(* Logix 5000 project; controller Safety vendor 1 type 14 code 86 rev 19.11; software revision 19.01; part 12 of 17 *)
(* tags used below, declared in another part *)
   A1_CoilCarSolPwrEn : BOOL;   // A1 UNW COIL CAR Solenoid Safe-Off Enable ( 1= Enable )
   A1_SolPwrEn : BOOL;   // A1 Solenoid Safe-Off Enable ( 1= Enable )
   A1_UnwLC_OK : BOOL;   // Unwind Light Curtain A/B ( 1= Not Blocked) ( 0= Blocked)
   A1_UnwLC_RstCmd : BOOL;   // Unwind Light Curtain Reset Command ( 1= Reset Cmd)
   C1_SolPwrEn : BOOL;   // C1 Solenoid Safe-Off Enable ( 1= Enable )
   CC_Toggle : DINT;   // TEST
   D1_SolPwrEn : BOOL;   // D1 Solenoid Safe-Off Enable ( 1= Enable )
   DPD_SolPwrEn : BOOL;   // DPD Solenoid Safe-Off Enable ( 1= Enable )
   E1_SolPwrEn : BOOL;   // E1 Solenoid Safe-Off Enable ( 1= Enable )
   Line_TotalMode : BOOL;   // Line TOTAL Mode ( 1= Total Mode) (0 = Coil to Coil)
   LineSts : UDT_SysStatus;
   OS4N_SolPwrEn : BOOL;   // OS4N Solenoid Safe-Off Enable ( 1= Enable )
   OS4S_SolPwrEn : BOOL;   // OS4S Solenoid Safe-Off Enable ( 1= Enable )
   PrCon_DrvsOff : BOOL;   // Product Conveyors (1-3) Drives OFF ( 1= OFF)
   PrCon_SafeTrqEn : BOOL;   // Product Conveyors Safe-Trq Off Enable ( 1= Enable )
   ScInCon_DrvsOff : BOOL;   // Scrap Incline Conveyor Drives OFF ( 1= OFF)
   ScInCon_SafeTrqEn : BOOL;   // Scrap Incline Conveyor Safe-Trq Off Enable ( 1= Enable )
   SDPLC_SolPwrEn : BOOL;   // SDPLC Solenoid Safe-Off Enable ( 1= Enable )
   ShearSts : UDT_ShearStatus;
   SkBkSt_DrvsOff : BOOL;   // Stacker Backstop Drives OFF ( 1= OFF)
   SkBkSt_SafeTrqEn : BOOL;   // Stacker Back Stop Safe-Trq Off Enable ( 1= Enable )
   SkBlwr_DrvsOff : BOOL;   // Stacker Blower Drives OFF ( 1= OFF)
   SkBlwr_SafeTrqEn : BOOL;   // Stacker Blower Safe-Trq Off Enable ( 1= Enable )
   Sr_DrvsOff : BOOL;   // Shear Pinch Roll/ Metering Back Up Drives OFF ( 1= OFF)
   Sr_SafeTrqEn : BOOL;   // Shear Pinch Roll/ Back Up Roll Safe-Trq Off Enable ( 1= Enable )
   SrCon_DrvsOff : BOOL;   // Shear Conveyor Drives OFF ( 1= OFF)
   SrCon_SafeTrqEn : BOOL;   // Shear Conveyor Safe-Trq Off Enable ( 1= Enable )
   StPR_DrvsOff : BOOL;   // Sheeter Pinch Roll Drives OFF ( 1= OFF)
   StPR_SafeTrqEn : BOOL;   // Sheeter Pinch Roll Safe-Trq Off Enable ( 1= Enable )
   UWCC_Rst_PB : ALIAS FOR SftyMap_Mach[0].10;   // Unwind Coil Car Safety Reset PB
   x406LCA047 : ALIAS FOR A1:21:I.Pt00Data;   // North/South Light Curtain Output A
   x406LCB052 : ALIAS FOR A1:21:I.Pt01Data;   // North/South Light Curtain Output B
   y172CR550 : ALIAS FOR SDPLC:2:O.Pt02Data;   // Line Soleniod Safe-Off
   y233CR040 : ALIAS FOR OS4N:5:O.Pt00Data;   // OS4N Solenoid Safe Off
   y243CR040 : ALIAS FOR OS4S:5:O.Pt00Data;   // OS4S Solenoid Safe Off
   y406CR050 : ALIAS FOR A1:20:O.Pt00Data;   // Line Solenoid Safe Off
   y406CR090 : ALIAS FOR A1:20:O.Pt01Data;   // Coil Car Solenoid Safe Off
   y435CR050 : ALIAS FOR C1:12:O.Pt00Data;   // Solenoid Safe Off
   y451CR050 : ALIAS FOR D1:12:O.Pt00Data;   // Soleniod Safe Off
   y464CR050 : ALIAS FOR E1:10:O.Pt00Data;   // Soleniod Safe Off
   y480CR050 : ALIAS FOR DPD:14:O.Pt00Data;   // Solenoid Safe Off
   y495CR050 : ALIAS FOR VS2:10:O.Pt00Data;   // Soleniod Safe Off
   y507CR090 : ALIAS FOR F1:19:O.Pt01Data;   // Rewind Coil Car Solenoid Safe Off
   y519CR050 : ALIAS FOR G1:11:O.Pt00Data;   // Line Solenoid Safe Off
   y533CR050 : ALIAS FOR H1:5:O.Pt00Data;   // Line Solenoid Safe Off
   y776MTR080SE : ALIAS FOR MCC4:3:O.Pt07Data;   // Shear Metering Backup Roll Safety Enable
   y776MTR080SP : ALIAS FOR MCC4:3:O.Pt06Data;   // Shear Metering Backup Roll Safety Power
   y779MTR080SE : ALIAS FOR MCC4:3:O.Pt01Data;   // Shear Pinch Roll Safety Enable
   y779MTR080SP : ALIAS FOR MCC4:3:O.Pt00Data;   // Shear Pinch Roll Safety Power
   y782MTR080SE : ALIAS FOR MCC4:3:O.Pt03Data;   // Sheeter Pinch Roll Safety Enable
   y782MTR080SP : ALIAS FOR MCC4:3:O.Pt02Data;   // Sheeter Pinch Roll Safety Power
   y785MTR080SE : ALIAS FOR MCC4:3:O.Pt05Data;   // Stacker Blower Safety Enable
   y785MTR080SP : ALIAS FOR MCC4:3:O.Pt04Data;   // Stacker Blower Safety Power
   y800MTR080SE : ALIAS FOR MCC5:3:O.Pt01Data;   // Scrap Incline Conveyor Safety Enable
   y800MTR080SP : ALIAS FOR MCC5:3:O.Pt00Data;   // Scrap Incline Conveyor Safety Power
   y804MTR080SE : ALIAS FOR MCC5:3:O.Pt03Data;   // Stacker Back Stop Safety Enable
   y804MTR080SP : ALIAS FOR MCC5:3:O.Pt02Data;   // Stacker Back Stop Safety Power
   y806MTR080SE : ALIAS FOR MCC5:3:O.Pt05Data;   // Product Conveyor 3 Safety Enable
   y806MTR080SP : ALIAS FOR MCC5:3:O.Pt04Data;   // Product Conveyor 3 Safety Power
   y808MTR080SE : ALIAS FOR MCC5:3:O.Pt07Data;   // Product Conveyor 1 Safety Enable
   y808MTR080SP : ALIAS FOR MCC5:3:O.Pt06Data;   // Product Conveyor 1 Safety Power
   y810MTR080SE : ALIAS FOR MCC5:4:O.Pt01Data;   // Product Conveyor 2 Safety Enable
   y810MTR080SP : ALIAS FOR MCC5:4:O.Pt00Data;   // Product Conveyor 2 Safety Power
   y812MTR080SE : ALIAS FOR MCC5:4:O.Pt03Data;   // Shear Conveyor Safety Enable
   y812MTR080SP : ALIAS FOR MCC5:4:O.Pt02Data;   // Shear Conveyor Safety Power
(* SafeOff, continued *)

ROUTINE B07_StPR_SafeTrqOff   (* ladder *)
// Sheeter Pinch Roll
// Safety Power Enable
// (Safe Trq Off and Drv Enable)
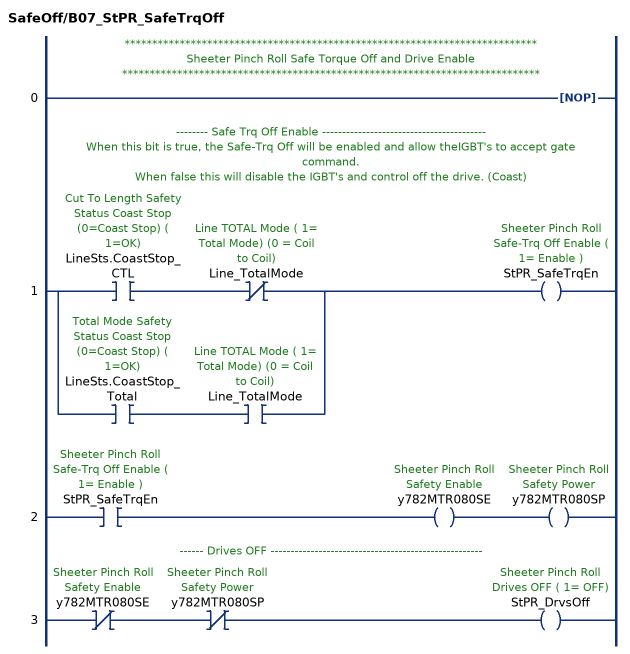
   // ***************************************************************************
   // Sheeter Pinch Roll Safe Torque Off and Drive Enable
   // ****************************************************************************
   0: NOP();
   // -------- Safe Trq Off Enable -----------------------------------------
   // When this bit is true, the Safe-Trq Off will be enabled and allow theIGBT's to accept gate command.
   // When false this will disable the IGBT's and control off the drive. (Coast)
   1: [XIC(LineSts.CoastStop_CTL) XIO(Line_TotalMode) ,XIC(LineSts.CoastStop_Total) XIC(Line_TotalMode) ]OTE(StPR_SafeTrqEn);
   2: XIC(StPR_SafeTrqEn)OTE(y782MTR080SE)OTE(y782MTR080SP);
   // ------ Drives OFF -----------------------------------------------------
   3: XIO(y782MTR080SE)XIO(y782MTR080SP)OTE(StPR_DrvsOff);
END_ROUTINE

ROUTINE B08_Sr_SafeTrqOff   (* ladder *)
// Sheear Pinch Roll /
// Back Up Metering
// Safety Power Enable
// (Safe Trq Off and Drv Enable)
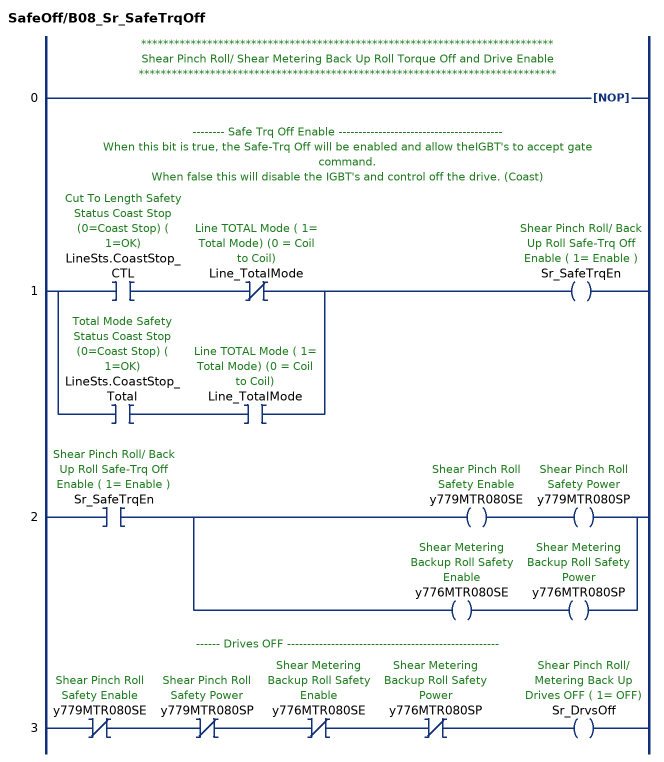
   // ***************************************************************************
   // Shear Pinch Roll/ Shear Metering Back Up Roll Torque Off and Drive Enable
   // ****************************************************************************
   0: NOP();
   // -------- Safe Trq Off Enable -----------------------------------------
   // When this bit is true, the Safe-Trq Off will be enabled and allow theIGBT's to accept gate command.
   // When false this will disable the IGBT's and control off the drive. (Coast)
   1: [XIC(LineSts.CoastStop_CTL) XIO(Line_TotalMode) ,XIC(LineSts.CoastStop_Total) XIC(Line_TotalMode) ]OTE(Sr_SafeTrqEn);
   2: XIC(Sr_SafeTrqEn)[OTE(y779MTR080SE) OTE(y779MTR080SP) ,OTE(y776MTR080SE) OTE(y776MTR080SP) ];
   // ------ Drives OFF -----------------------------------------------------
   3: XIO(y779MTR080SE)XIO(y779MTR080SP)XIO(y776MTR080SE)XIO(y776MTR080SP)OTE(Sr_DrvsOff);
END_ROUTINE

ROUTINE B09_SrCon_SafeTrqOff   (* ladder *)
// Shear Conveyor
// Safety Power Enable
// (Safe Trq Off and Drv Enable)
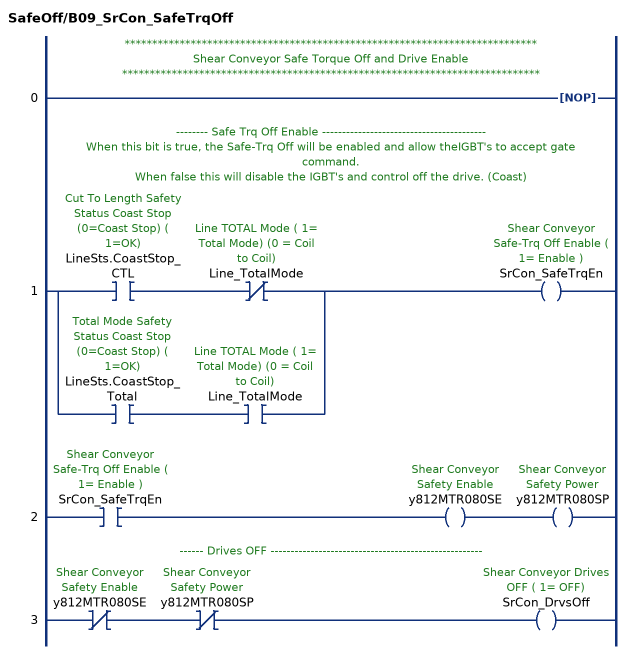
   // ***************************************************************************
   // Shear Conveyor Safe Torque Off and Drive Enable
   // ****************************************************************************
   0: NOP();
   // -------- Safe Trq Off Enable -----------------------------------------
   // When this bit is true, the Safe-Trq Off will be enabled and allow theIGBT's to accept gate command.
   // When false this will disable the IGBT's and control off the drive. (Coast)
   1: [XIC(LineSts.CoastStop_CTL) XIO(Line_TotalMode) ,XIC(LineSts.CoastStop_Total) XIC(Line_TotalMode) ]OTE(SrCon_SafeTrqEn);
   2: XIC(SrCon_SafeTrqEn)OTE(y812MTR080SE)OTE(y812MTR080SP);
   // ------ Drives OFF -----------------------------------------------------
   3: XIO(y812MTR080SE)XIO(y812MTR080SP)OTE(SrCon_DrvsOff);
END_ROUTINE

ROUTINE B10_PrCon_SafeTrqOff   (* ladder *)
// Product Conveyors (1-3)
// Safety Power Enable
// (Safe Trq Off and Drv Enable)
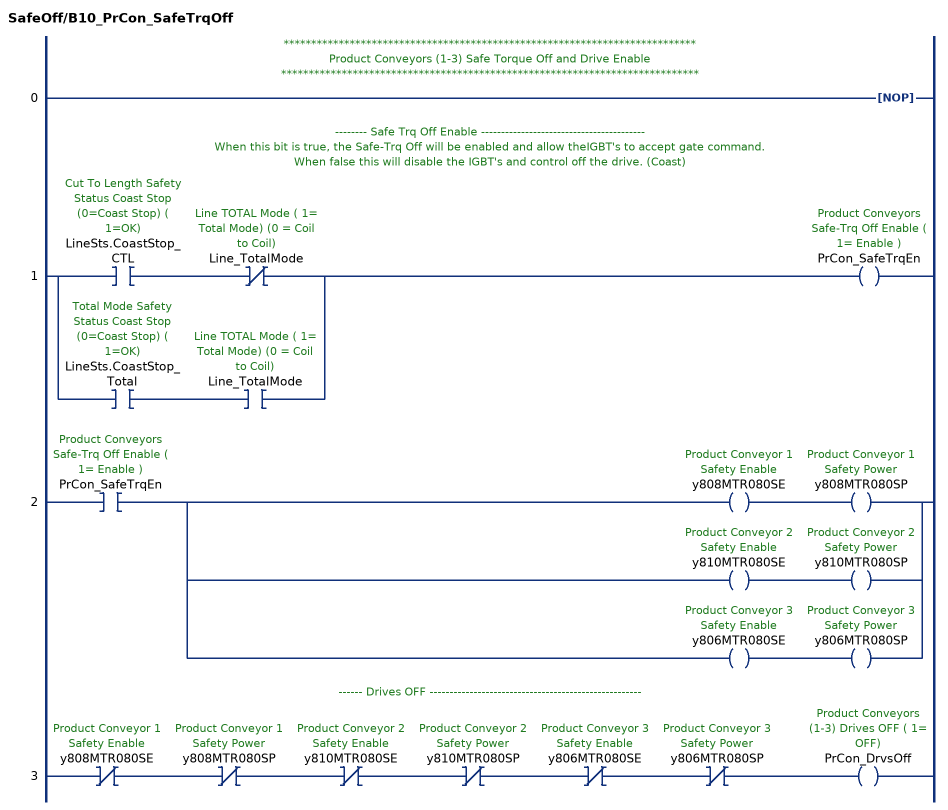
   // ***************************************************************************
   // Product Conveyors (1-3) Safe Torque Off and Drive Enable
   // ****************************************************************************
   0: NOP();
   // -------- Safe Trq Off Enable -----------------------------------------
   // When this bit is true, the Safe-Trq Off will be enabled and allow theIGBT's to accept gate command.
   // When false this will disable the IGBT's and control off the drive. (Coast)
   1: [XIC(LineSts.CoastStop_CTL) XIO(Line_TotalMode) ,XIC(LineSts.CoastStop_Total) XIC(Line_TotalMode) ]OTE(PrCon_SafeTrqEn);
   2: XIC(PrCon_SafeTrqEn)[OTE(y808MTR080SE) OTE(y808MTR080SP) ,OTE(y810MTR080SE) OTE(y810MTR080SP) ,OTE(y806MTR080SE) OTE(y806MTR080SP) ];
   // ------ Drives OFF -----------------------------------------------------
   3: XIO(y808MTR080SE)XIO(y808MTR080SP)XIO(y810MTR080SE)XIO(y810MTR080SP)XIO(y806MTR080SE)XIO(y806MTR080SP)OTE(PrCon_DrvsOff);
END_ROUTINE

ROUTINE B11_ScIncCon_SafeTrqOff   (* ladder *)
// Scrap Incline Conveyor
// Safety Power Enable
// (Safe Trq Off and Drv Enable)
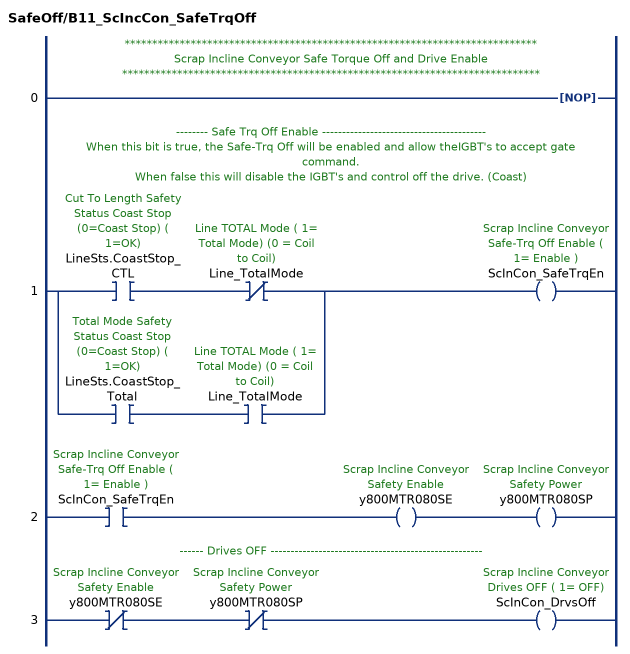
   // ***************************************************************************
   // Scrap Incline Conveyor Safe Torque Off and Drive Enable
   // ****************************************************************************
   0: NOP();
   // -------- Safe Trq Off Enable -----------------------------------------
   // When this bit is true, the Safe-Trq Off will be enabled and allow theIGBT's to accept gate command.
   // When false this will disable the IGBT's and control off the drive. (Coast)
   1: [XIC(LineSts.CoastStop_CTL) XIO(Line_TotalMode) ,XIC(LineSts.CoastStop_Total) XIC(Line_TotalMode) ]OTE(ScInCon_SafeTrqEn);
   2: XIC(ScInCon_SafeTrqEn)OTE(y800MTR080SE)OTE(y800MTR080SP);
   // ------ Drives OFF -----------------------------------------------------
   3: XIO(y800MTR080SE)XIO(y800MTR080SP)OTE(ScInCon_DrvsOff);
END_ROUTINE

ROUTINE B12_SkBlwr_SafeTrqOff   (* ladder *)
// Stacker Blower
// Safety Power Enable
// (Safe Trq Off and Drv Enable)
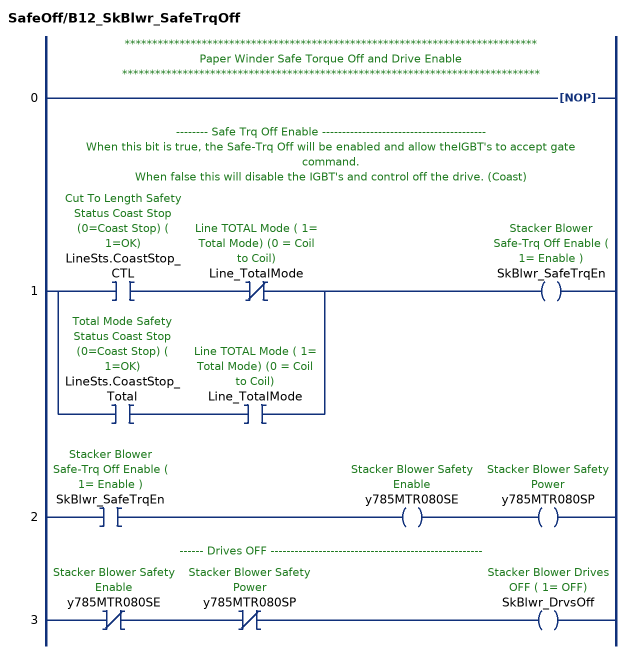
   // ***************************************************************************
   // Paper Winder Safe Torque Off and Drive Enable
   // ****************************************************************************
   0: NOP();
   // -------- Safe Trq Off Enable -----------------------------------------
   // When this bit is true, the Safe-Trq Off will be enabled and allow theIGBT's to accept gate command.
   // When false this will disable the IGBT's and control off the drive. (Coast)
   1: [XIC(LineSts.CoastStop_CTL) XIO(Line_TotalMode) ,XIC(LineSts.CoastStop_Total) XIC(Line_TotalMode) ]OTE(SkBlwr_SafeTrqEn);
   2: XIC(SkBlwr_SafeTrqEn)OTE(y785MTR080SE)OTE(y785MTR080SP);
   // ------ Drives OFF -----------------------------------------------------
   3: XIO(y785MTR080SE)XIO(y785MTR080SP)OTE(SkBlwr_DrvsOff);
END_ROUTINE

ROUTINE B13_SkBkSt_SafeTrqOff   (* ladder *)
// Stacker Back Stop
// Safety Power Enable
// (Safe Trq Off and Drv Enable)
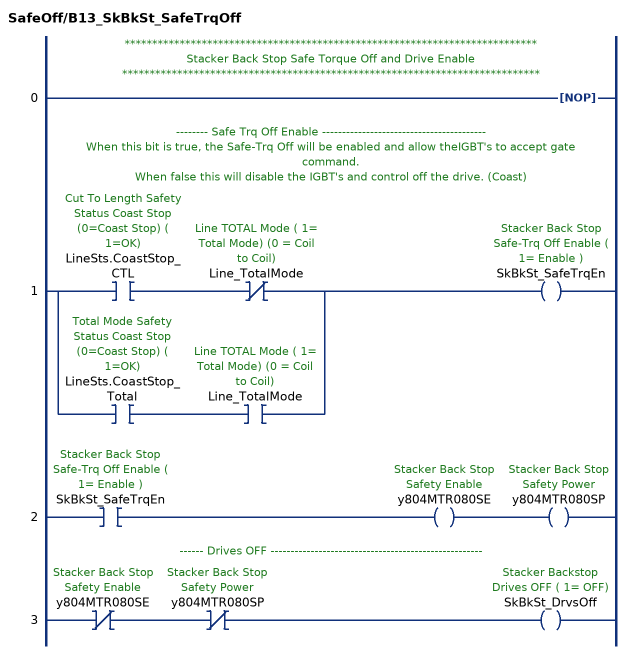
   // ***************************************************************************
   // Stacker Back Stop Safe Torque Off and Drive Enable
   // ****************************************************************************
   0: NOP();
   // -------- Safe Trq Off Enable -----------------------------------------
   // When this bit is true, the Safe-Trq Off will be enabled and allow theIGBT's to accept gate command.
   // When false this will disable the IGBT's and control off the drive. (Coast)
   1: [XIC(LineSts.CoastStop_CTL) XIO(Line_TotalMode) ,XIC(LineSts.CoastStop_Total) XIC(Line_TotalMode) ]OTE(SkBkSt_SafeTrqEn);
   2: XIC(SkBkSt_SafeTrqEn)OTE(y804MTR080SE)OTE(y804MTR080SP);
   // ------ Drives OFF -----------------------------------------------------
   3: XIO(y804MTR080SE)XIO(y804MTR080SP)OTE(SkBkSt_DrvsOff);
END_ROUTINE
END_PROGRAM

PROGRAM Safety_JUNK   (* main routine Scratch *)

ROUTINE Scratch   (* ladder *)
   0: NOP();
END_ROUTINE
END_PROGRAM

PROGRAM Solenoid_Pwr   (* main routine A00_Main *)
// Control fo the Field Power
// to the Solenoids

ROUTINE A00_Main   (* ladder *)
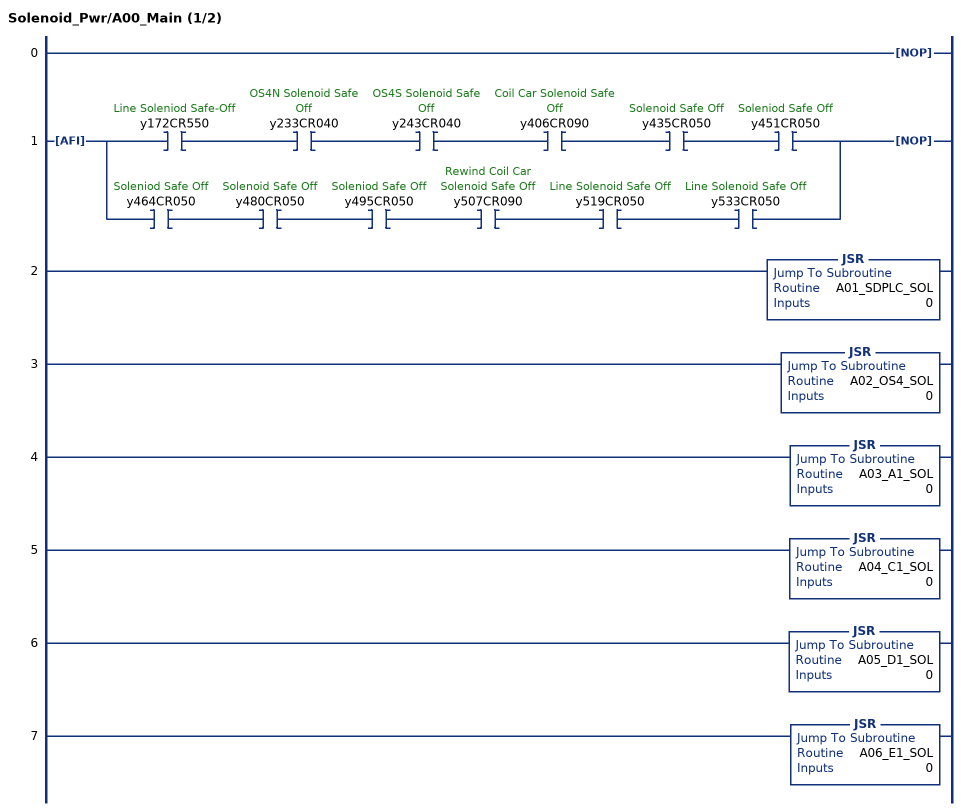
   0: NOP();
   1: AFI()[XIC(y172CR550) XIC(y233CR040) XIC(y243CR040) XIC(y406CR090) XIC(y435CR050) XIC(y451CR050) ,XIC(y464CR050) XIC(y480CR050) XIC(y495CR050) XIC(y507CR090) XIC(y519CR050) XIC(y533CR050) ]NOP();
   2: JSR(A01_SDPLC_SOL,0);
   3: JSR(A02_OS4_SOL,0);
   4: JSR(A03_A1_SOL,0);
   5: JSR(A04_C1_SOL,0);
   6: JSR(A05_D1_SOL,0);
   7: JSR(A06_E1_SOL,0);
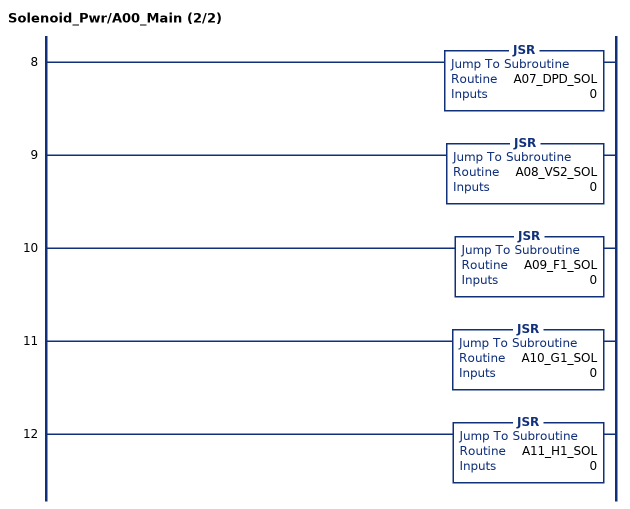
   8: JSR(A07_DPD_SOL,0);
   9: JSR(A08_VS2_SOL,0);
   10: JSR(A09_F1_SOL,0);
   11: JSR(A10_G1_SOL,0);
   12: JSR(A11_H1_SOL,0);
END_ROUTINE

ROUTINE A01_SDPLC_SOL   (* ladder *)
// SDPLC
// Solenoid Power Enable
// (FPD Power Removal)
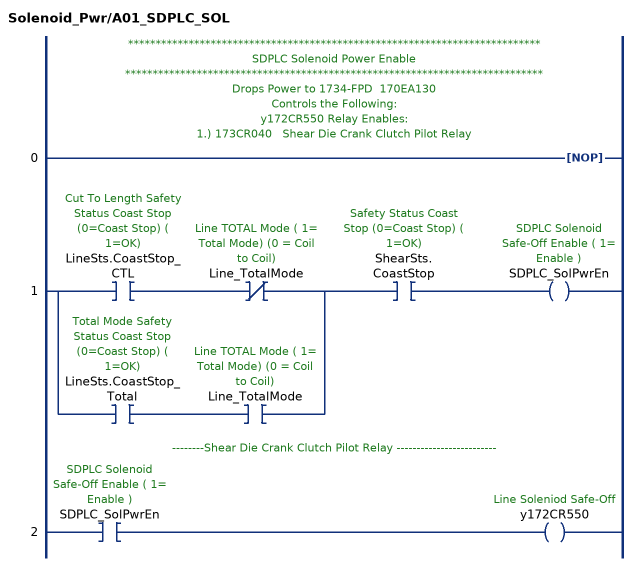
   // ***************************************************************************
   // SDPLC Solenoid Power Enable
   // ****************************************************************************
   // Drops Power to 1734-FPD	170EA130
   // Controls the Following:
   // y172CR550 Relay Enables:
   // 1.) 173CR040   Shear Die Crank Clutch Pilot Relay
   0: NOP();
   1: [XIC(LineSts.CoastStop_CTL) XIO(Line_TotalMode) ,XIC(LineSts.CoastStop_Total) XIC(Line_TotalMode) ]XIC(ShearSts.CoastStop)OTE(SDPLC_SolPwrEn);
   // --------Shear Die Crank Clutch Pilot Relay -------------------------
   2: XIC(SDPLC_SolPwrEn)OTE(y172CR550);
END_ROUTINE

ROUTINE A02_OS4_SOL   (* ladder *)
// OS4N/S
// Solenoid Power Enable
// (FPD Power Removal)
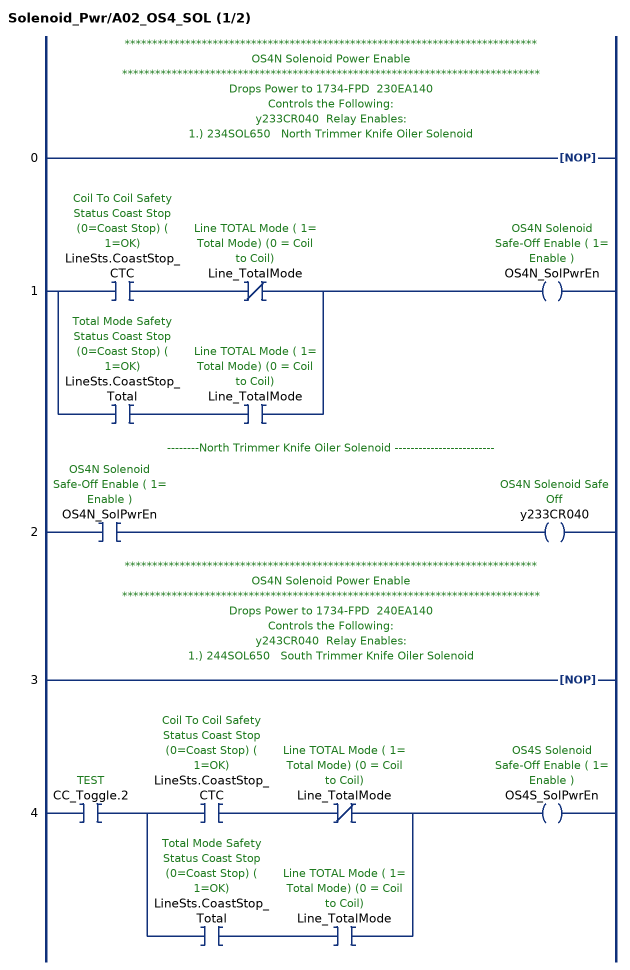
   // ***************************************************************************
   // OS4N Solenoid Power Enable
   // ****************************************************************************
   // Drops Power to 1734-FPD	230EA140
   // Controls the Following:
   // y233CR040  Relay Enables:
   // 1.) 234SOL650   North Trimmer Knife Oiler Solenoid
   0: NOP();
   1: [XIC(LineSts.CoastStop_CTC) XIO(Line_TotalMode) ,XIC(LineSts.CoastStop_Total) XIC(Line_TotalMode) ]OTE(OS4N_SolPwrEn);
   // --------North Trimmer Knife Oiler Solenoid -------------------------
   2: XIC(OS4N_SolPwrEn)OTE(y233CR040);
   // ***************************************************************************
   // OS4N Solenoid Power Enable
   // ****************************************************************************
   // Drops Power to 1734-FPD	240EA140
   // Controls the Following:
   // y243CR040  Relay Enables:
   // 1.) 244SOL650   South Trimmer Knife Oiler Solenoid
   3: NOP();
   4: XIC(CC_Toggle.2)[XIC(LineSts.CoastStop_CTC) XIO(Line_TotalMode) ,XIC(LineSts.CoastStop_Total) XIC(Line_TotalMode) ]OTE(OS4S_SolPwrEn);
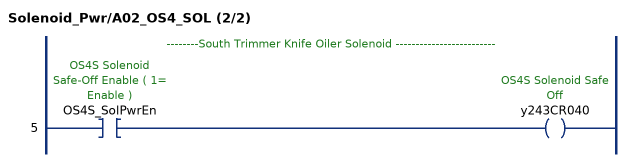
   // --------South Trimmer Knife Oiler Solenoid -------------------------
   5: XIC(OS4S_SolPwrEn)OTE(y243CR040);
END_ROUTINE

ROUTINE A03_A1_SOL   (* ladder *)
// A1
// Solenoid Power Enable
// (FPD Power Removal)
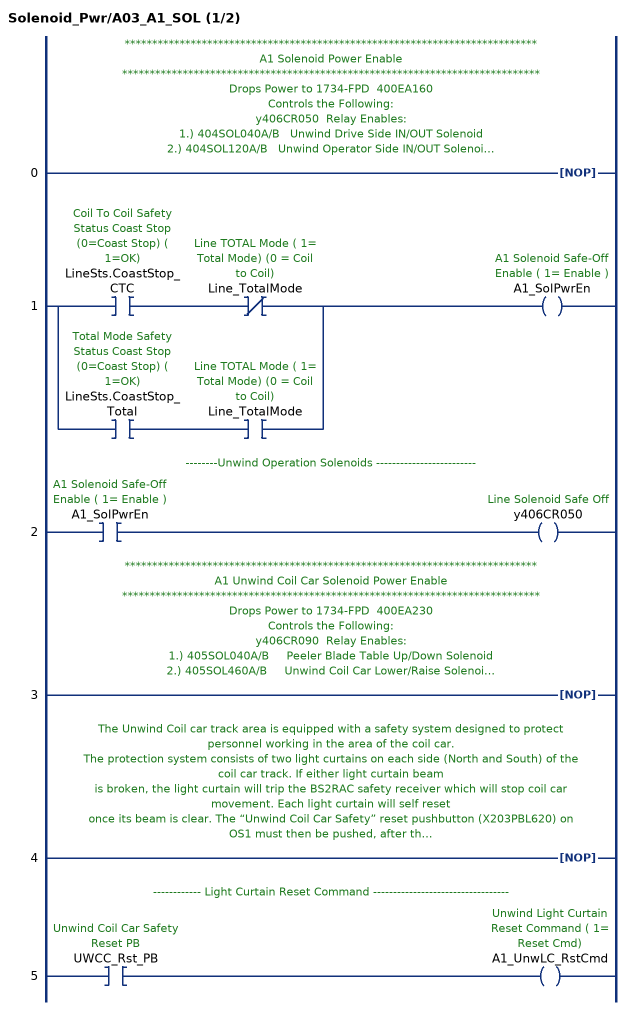
   // ***************************************************************************
   // A1 Solenoid Power Enable
   // ****************************************************************************
   // Drops Power to 1734-FPD	400EA160
   // Controls the Following:
   // y406CR050  Relay Enables:
   // 1.) 404SOL040A/B   Unwind Drive Side IN/OUT Solenoid
   // 2.) 404SOL120A/B   Unwind Operator Side IN/OUT Solenoid
   // 3.) 404SOL220A/B   Unwind Reel Tandem North Solenoid
   // 4.) 404SOL300         Unwind Reel Tandem Unlock Solenoid
   // 5.) 404SOL460A      Unwind Hold Down Roll Lower/Raise Solenoid
   // 6.) 404SOL640A/B   Unwind Peeler Blade Extend/Retract Solenoid
   // 7.) 404SOL680A/B   Unwind Peeler Blade Pivot Lower/Raise Solenoid
   0: NOP();
   1: [XIC(LineSts.CoastStop_CTC) XIO(Line_TotalMode) ,XIC(LineSts.CoastStop_Total) XIC(Line_TotalMode) ]OTE(A1_SolPwrEn);
   // --------Unwind Operation Solenoids -------------------------
   2: XIC(A1_SolPwrEn)OTE(y406CR050);
   // ***************************************************************************
   // A1 Unwind Coil Car Solenoid Power Enable
   // ****************************************************************************
   // Drops Power to 1734-FPD	400EA230
   // Controls the Following:
   // y406CR090  Relay Enables:
   // 1.) 405SOL040A/B     Peeler Blade Table Up/Down Solenoid
   // 2.) 405SOL460A/B     Unwind Coil Car Lower/Raise Solenoid
   // 3.) 405SOL540A/B     Unwind Coil Car Traverse IN/OUT Solenoid
   3: NOP();
   // The Unwind Coil car track area is equipped with a safety system designed to protect personnel working in the area of the coil car.
   // The protection system consists of two light curtains on each side (North and South) of the coil car track. If either light curtain beam
   // is broken, the light curtain will trip the BS2RAC safety receiver which will stop coil car movement. Each light curtain will self reset
   //  once its beam is clear. The “Unwind Coil Car Safety” reset pushbutton (X203PBL620) on OS1 must then be pushed, after the
   // area has been cleared, to reset the system and allow the coil car to continue movement.
   4: NOP();
   // ------------ Light Curtain Reset Command ----------------------------------
   5: XIC(UWCC_Rst_PB)OTE(A1_UnwLC_RstCmd);
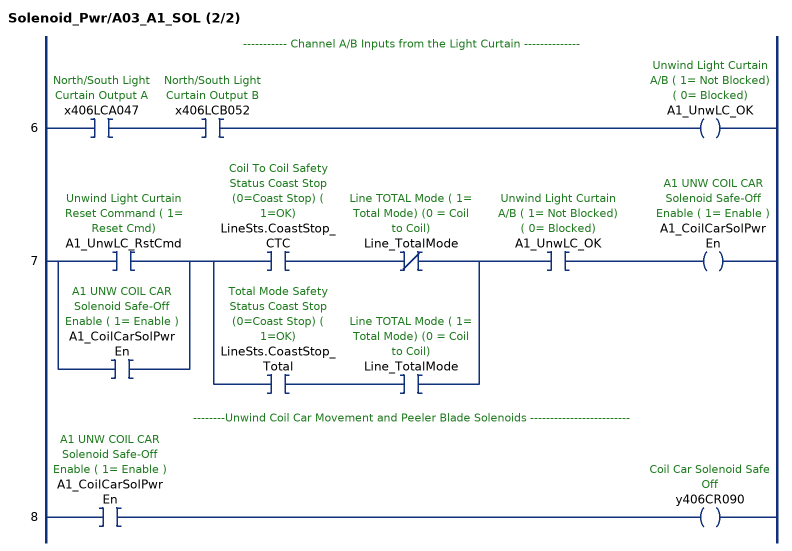
   // ----------- Channel A/B Inputs from the Light Curtain --------------
   6: XIC(x406LCA047)XIC(x406LCB052)OTE(A1_UnwLC_OK);
   7: [XIC(A1_UnwLC_RstCmd) ,XIC(A1_CoilCarSolPwrEn) ][XIC(LineSts.CoastStop_CTC) XIO(Line_TotalMode) ,XIC(LineSts.CoastStop_Total) XIC(Line_TotalMode) ]XIC(A1_UnwLC_OK)OTE(A1_CoilCarSolPwrEn);
   // --------Unwind Coil Car Movement and Peeler Blade Solenoids -------------------------
   8: XIC(A1_CoilCarSolPwrEn)OTE(y406CR090);
END_ROUTINE

ROUTINE A04_C1_SOL   (* ladder *)
// C1
// Solenoid Power Enable
// (FPD Power Removal)
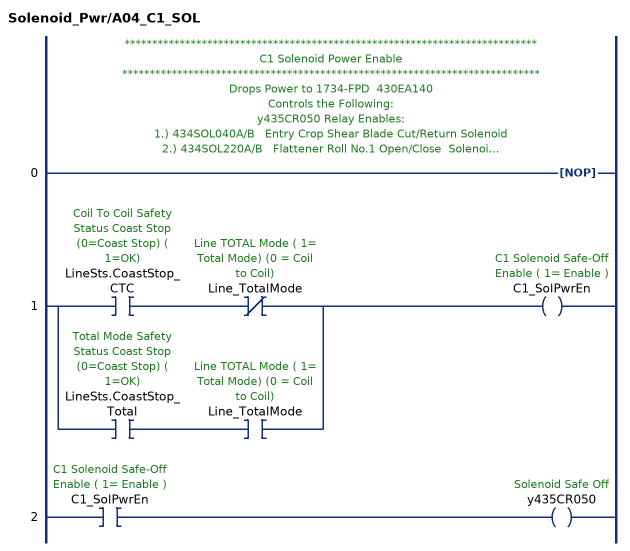
   // ***************************************************************************
   // C1 Solenoid Power Enable
   // ****************************************************************************
   // Drops Power to 1734-FPD	430EA140
   // Controls the Following:
   // y435CR050 Relay Enables:
   // 1.) 434SOL040A/B   Entry Crop Shear Blade Cut/Return Solenoid
   // 2.) 434SOL220A/B   Flattener Roll No.1 Open/Close  Solenoid
   // 3.) 434SOL300A/B   Flattener Roll No.2 Open/Close  Solenoid
   // 4.) 434SOL460A/B  Side Guide Quick Close/Open Solenoid
   0: NOP();
   1: [XIC(LineSts.CoastStop_CTC) XIO(Line_TotalMode) ,XIC(LineSts.CoastStop_Total) XIC(Line_TotalMode) ]OTE(C1_SolPwrEn);
   2: XIC(C1_SolPwrEn)OTE(y435CR050);
END_ROUTINE

ROUTINE A05_D1_SOL   (* ladder *)
// D1
// Solenoid Power Enable
// (FPD Power Removal)
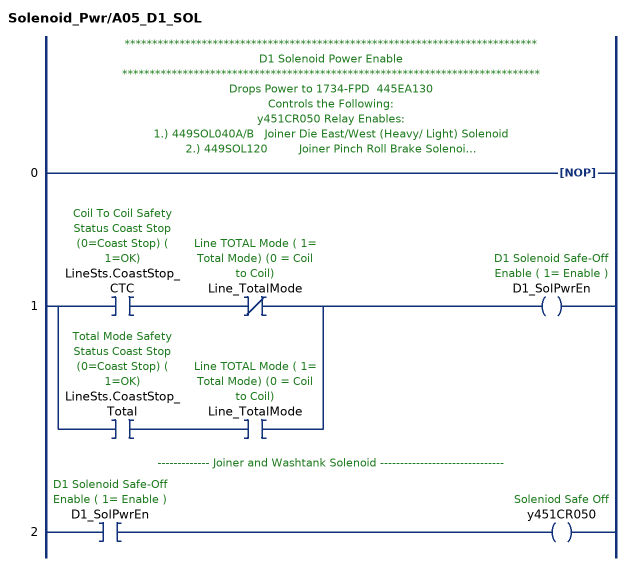
   // ***************************************************************************
   // D1 Solenoid Power Enable
   // ****************************************************************************
   // Drops Power to 1734-FPD	445EA130
   // Controls the Following:
   // y451CR050 Relay Enables:
   // 1.) 449SOL040A/B   Joiner Die East/West (Heavy/ Light) Solenoid
   // 2.) 449SOL120         Joiner Pinch Roll Brake Solenoid
   // 3.) 449SOL220A/B   Joiner Press/Raise  Solenoid
   // 4.) 449SOL300         Joiner Relief Solenoid
   // 5.) 449SOL460        Wash Tank Pinch Roll 1 Open Solenoid
   // 6.) 449SOL500        Wash Tank Pinch Roll 2 Open Solenoid
   // 7.) 449SOL540        Wash Tank Pinch Roll 3 Open Solenoid
   // 8.) 449SOL580        Wash Tank Pinch Roll 4 Open Solenoid
   0: NOP();
   1: [XIC(LineSts.CoastStop_CTC) XIO(Line_TotalMode) ,XIC(LineSts.CoastStop_Total) XIC(Line_TotalMode) ]OTE(D1_SolPwrEn);
   // ------------- Joiner and Washtank Solenoid -------------------------------
   2: XIC(D1_SolPwrEn)OTE(y451CR050);
END_ROUTINE

ROUTINE A06_E1_SOL   (* ladder *)
// E1
// Solenoid Power Enable
// (FPD Power Removal)
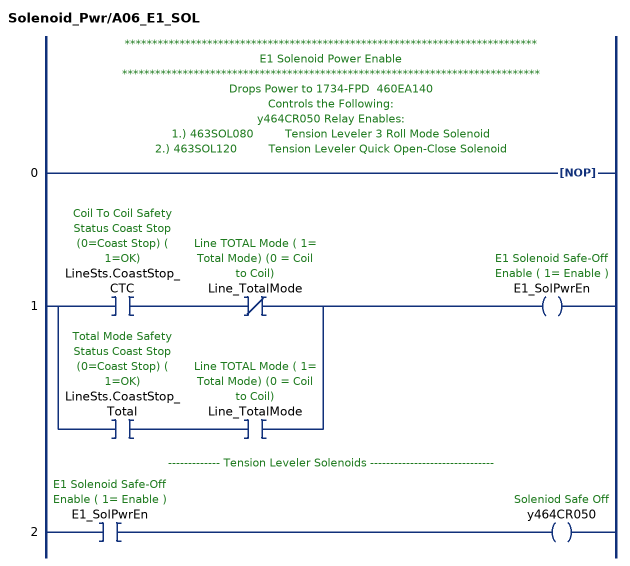
   // ***************************************************************************
   // E1 Solenoid Power Enable
   // ****************************************************************************
   // Drops Power to 1734-FPD	460EA140
   // Controls the Following:
   // y464CR050 Relay Enables:
   // 1.) 463SOL080         Tension Leveler 3 Roll Mode Solenoid
   // 2.) 463SOL120         Tension Leveler Quick Open-Close Solenoid
   0: NOP();
   1: [XIC(LineSts.CoastStop_CTC) XIO(Line_TotalMode) ,XIC(LineSts.CoastStop_Total) XIC(Line_TotalMode) ]OTE(E1_SolPwrEn);
   // ------------- Tension Leveler Solenoids -------------------------------
   2: XIC(E1_SolPwrEn)OTE(y464CR050);
END_ROUTINE

ROUTINE A07_DPD_SOL   (* ladder *)
// DPD
// Solenoid Power Enable
// (FPD Power Removal)
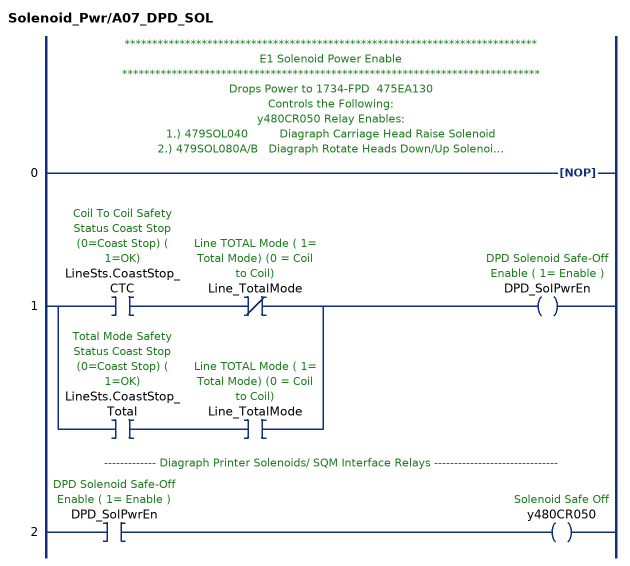
   // ***************************************************************************
   // E1 Solenoid Power Enable
   // ****************************************************************************
   // Drops Power to 1734-FPD	475EA130
   // Controls the Following:
   // y480CR050 Relay Enables:
   // 1.) 479SOL040         Diagraph Carriage Head Raise Solenoid
   // 2.) 479SOL080A/B   Diagraph Rotate Heads Down/Up Solenoid
   // 3.) 479SOL220         Marker Safety Gate Solenoid
   // 4.) 479CR300           SQM Next Inspection Relay
   // 5.) 479CR340           SQM Reserved Relay
   0: NOP();
   1: [XIC(LineSts.CoastStop_CTC) XIO(Line_TotalMode) ,XIC(LineSts.CoastStop_Total) XIC(Line_TotalMode) ]OTE(DPD_SolPwrEn);
   // ------------- Diagraph Printer Solenoids/ SQM Interface Relays -------------------------------
   2: XIC(DPD_SolPwrEn)OTE(y480CR050);
END_ROUTINE
